Universal Robots PolyScope program: DynamicCartesianPositionCheck.urp

ProgramRoot directory=/home/ur/ursim-3.1/programs/Howtos; kinematics=(a=[0, -0.425, -0.39225, 0, 0, 0], d=[0.08916, 0, 0, 0.10915, 0.09465, 0.0823], alpha=[1.5708, 0, 0, 1.5708, -1.5708, 0], deltaTheta=[0, 0, 0, 0, 0, 0], status=notInitialized); lastSavedInVersion=(project__name=Polyscope, major__version=3, minor__version=1, svn__revision=17195, build__date=Mar 11 2015, 13:02:28); name=DynamicCartesianPositionCheck; programVersion=(project__name=Polyscope, major__version=3, minor__version=1, svn__revision=17195, build__date=Mar 11 2015, 13:02:28); robotEnvironmentFileName=default; serialNumberRobot=2014350001
  MainProgram cartesianAcceleration=1.2; cartesianSpeed=0.25; jointAcceleration=1.3962634015954636; jointSpeed=1.0471975511965976; sharedProcessMoveBlendRadius=0.025; motionType=JOINT_SPACE
    Move cartesianAcceleration=1.2; cartesianSpeed=0.25; jointAcceleration=1.3962634015954636; jointSpeed=1.0471975511965976; sharedProcessMoveBlendRadius=0.025; motionType=CARTESIAN_SPACE
      Waypoint blendRadius=0.05; cartesianAcceleration=1.2; cartesianSpeed=0.25; jointAcceleration=1.3962634015954636; jointSpeed=1.0471975511965976; nextMotionTime=2.0; stoppoint=true; useSharedBlendParameter=true; useSharedParameters=true; outputFlangePose=(pos=(x=0.2455654667221236, y=0.04814591292354345, z=0.14607257413085825), rot=(x=2.594945247174466, y=-1.7582887050933431, z=-0.05448387356252551)); position=TCP in base x=245.565 y=48.146 z=146.073 mm, rx=2.5949 ry=-1.7583 rz=-0.0545 rad; joints [36.315, -66.39, -152.935, -51.698, 91.75, 14.541] deg; positionType=FIXED_POSITION; waypointPoseInFeatureCoordinates=(pos=(x=0.24556546619680325, y=0.0481459129235117, z=0.14607257413079386), rot=(x=2.594945247174335, y=-1.7582887050933247, z=-0.05448387356254208)); name=Waypoint_1
      Waypoint blendRadius=0.05; cartesianAcceleration=1.2; cartesianSpeed=0.25; jointAcceleration=1.3962634015954636; jointSpeed=1.0471975511965976; nextMotionTime=2.0; stoppoint=true; useSharedBlendParameter=true; useSharedParameters=true; outputFlangePose=(pos=(x=0.44556545731669017, y=0.04814591463289413, z=0.246072522914777), rot=(x=2.594945153378495, y=-1.7582886548687453, z=-0.054484026093422004)); position=TCP in base x=445.565 y=48.146 z=246.073 mm, rx=2.5949 ry=-1.7583 rz=-0.0545 rad; joints [20, -89.449, -118.424, -63.6, 91.393, -1.776] deg; positionType=FIXED_POSITION; waypointPoseInFeatureCoordinates=(pos=(x=0.4455654573166901, y=0.04814591463289411, z=0.24607252291477702), rot=(x=2.594945153378557, y=-1.7582886548687837, z=-0.05448402609345492)); name=Waypoint_2
  Thread name=Thread_1
    Assignment expr=get_actual_tcp_pose(); operatorValueType=INTEGER; valueSource=EXPRESSION
    Assignment expr=ExpressionVariableNode[0]; operatorValueType=INTEGER; valueSource=EXPRESSION
    Assignment expr=ExpressionVariableNode[2]; operatorValueType=INTEGER; valueSource=EXPRESSION
    If expr=(ExpressionVariableNode>0.3) and (ExpressionVariableNode>0.2); type=IF_NODE
      Set 
    If type=ELSE_NODE
      Set 
    Script type=0; expressionBranchNode=sync()
